FUNCTION F_GetTaskContext : I_ContextBuilder

F_GetTaskContext := GlobalVariables.aTaskLogger[GETCURTASKINDEXEX()].TaskContext;

END_FUNCTION

(* stored: Version 1.1.0.1, ProductVersion 3.1.4024.0
   POU F_GetTaskContext: Id {4f3df61f-e1b2-43bf-8e23-325425960015}, SpecialFunc None *)
